// TwinCAT 3 PLC project FMS_201_Estructurado
// ProgramVersion: 3.1.4024.0
// libraries:
//   Tc2_Standard, * (Beckhoff Automation GmbH)
//   Tc2_System, * (Beckhoff Automation GmbH)
//   Tc3_Module, * (Beckhoff Automation GmbH)
// project tree:
//   / PlcTask.TcTTO
//   POUs/Estación/ FB_Coordinador_SFC.TcPOU, FB_Estacion_SFC.TcPOU
//   POUs/ MAIN.TcPOU (not stored)
//   POUs/Tareas/ FB_2_AlimentarBase_SFC.TcPOU (not stored), FB_1_CargarBase_SFC.TcPOU, FB_4_InsertarBasePale_SFCC.TcPOU, FB_5_TransferirBase_SFC.TcPOU, FB_3_VerificarPale_SFC.TcPOU
// (motion and I/O tree: see PLC project fms_201_manual)
// real-time tasks:
//   TASK PlcTask: cycle T#10ms, priority 20, ADS port 350
//   TASK PlcTask1: cycle T#10ms, priority 21, ADS port 351
//   TASK PlcTask2: cycle T#10ms, priority 22, ADS port 352
// variable links:

CONFIGURATION FMS_201_Estructurado
    RESOURCE PLC ON TwinCAT3
        TASK PlcTask(INTERVAL := T#10ms, PRIORITY := 21);
        PROGRAM MAIN WITH PlcTask : MAIN;
    END_RESOURCE
END_CONFIGURATION

// ---- POUs/Estación/FB_Coordinador_SFC.TcPOU
FUNCTION_BLOCK FB_Coordinador_SFC
VAR_INPUT
END_VAR
VAR_OUTPUT
END_VAR
VAR
END_VAR

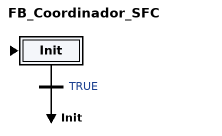
INITIAL_STEP Init:
END_STEP
TRANSITION FROM Init TO Init
    := TRUE;
END_TRANSITION

END_FUNCTION_BLOCK

// ---- POUs/Estación/FB_Estacion_SFC.TcPOU
FUNCTION_BLOCK FB_Estacion_SFC
VAR_INPUT
	// SFC-Flags
	SFCReset: BOOL;
	
	// Parámetros
	TpoEstabilidad: TIME := T#1000MS;
	UdsSolicitadas:UINT := 5;
	
END_VAR
VAR_OUTPUT
	// Parámetros
	CondicionInicial: BOOL;
	UdsPendientes: UINT;
	UdsRealizadas: BOOL;
	
	// Entradas comunes
	PulsadorEmergencia AT %I*: BOOL;
    SelectorManual AT %I*: BOOL;
    PulsadorMarcha AT %I*: BOOL;
    PulsadorParada AT %I*: BOOL := TRUE; // Contacto normalmente cerrado
    EstacionConectada AT %I*: BOOL := TRUE;
    DetectorPresion AT %I*: BOOL := TRUE;
	
	PalePresencia AT %I*: BOOL;
    PaleCodigoBit0 AT %I*: BOOL;
    PaleCodigoBit1 AT %I*: BOOL;
    PaleCodigoBit2 AT %I*: BOOL;
	
	// Entradas específicas
	DescargadorDetras AT %I*: BOOL;
	DescargadorDelante AT %I*: BOOL;
	VerticalArriba AT %I*: BOOL;
	VerticalAbajo AT %I*: BOOL;
	VerificadorArriba AT %I*: BOOL;
	VerificadorAbajo AT %I*: BOOL;
	DesplazadorDetras AT %I*: BOOL;
	AlimentadorDetras AT %I*: BOOL;
	AlimentadorDelante AT %I*: BOOL;
	VacioDescargador AT %I*: BOOL;
	PresenciaBaseAlimentador AT %I*:BOOL;
END_VAR
VAR
	// Bloques funcionales
	CLK: FB_Clock;
	// Salidas comunes
	DesconectaEstacion AT %Q*: BOOL;
    LamparaAlarma AT %Q*: BOOL;
    LamparaMarcha AT %Q*: BOOL;
	LamparaFaltaMaterial AT %Q*: BOOL;
    AvisadorSonoro AT %Q*: BOOL;

    CintaMotorActiva AT %Q*: BOOL;
    CintaMotorInvierte AT %Q*: BOOL;
    CintaRetenedorBaja AT %Q*: BOOL;
    CintaSeparadorSube AT %Q*: BOOL;
	
	// Salidas específicas
	DescargadorAtras AT %Q*: BOOL;
	DescargadorAdelante AT %Q*: BOOL;
	DescargadorBaja AT %Q*: BOOL;
	RechazadorAdelante AT %Q*: BOOL;
	VerificadorBaja AT %Q*: BOOL;
	DesplazadorAdelante AT %Q*: BOOL;
	AlimentadorAdelante AT %Q*: BOOL;
	EyectorSucciona AT %Q*: BOOL;
END_VAR

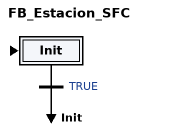
INITIAL_STEP Init:
END_STEP
TRANSITION FROM Init TO Init
    := TRUE;
END_TRANSITION

END_FUNCTION_BLOCK

// ---- POUs/Tareas/FB_1_CargarBase_SFC.TcPOU
FUNCTION_BLOCK FB_1_CargarBase_SFC
VAR_INPUT
	
	// Indicadores de sincronización
	Ack: BOOL := TRUE;
	Execute: BOOL;
	
	// Entradas
	PalePresencia AT %I*: BOOL;
	
END_VAR
VAR_OUTPUT
	
	// Indicadores de sincronización
	Ready: BOOL;	
	Done: BOOL;
	
	// Salidas
	CintaMotorActiva AT %Q*: BOOL;
	
END_VAR
VAR
END_VAR

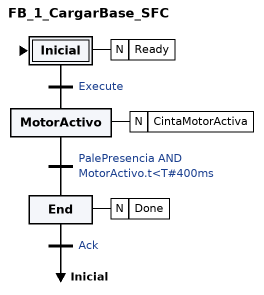
INITIAL_STEP Inicial:
    Ready(N);
END_STEP
TRANSITION FROM Inicial TO MotorActivo
    := Execute;
END_TRANSITION
STEP MotorActivo:
    CintaMotorActiva(N);
END_STEP
TRANSITION FROM MotorActivo TO End
    := PalePresencia AND MotorActivo.t<T#400ms;
END_TRANSITION
STEP End:
    Done(N);
END_STEP
TRANSITION FROM End TO Inicial
    := Ack;
END_TRANSITION

END_FUNCTION_BLOCK

// ---- POUs/Tareas/FB_4_InsertarBasePale_SFCC.TcPOU
FUNCTION_BLOCK FB_4_InsertarBasePale_SFCC
VAR_INPUT

// Indicadores de sincronización
	Ack: BOOL := TRUE;
	Execute: BOOL;
	
	// Parámetros
	TpoTraspase: TIME := T#500MS;
	
	// Entradas
	VerticalArriba AT %I*: BOOL;
	VerticalAbajo AT %I*: BOOL;
	VacioDescargador AT %I*: BOOL;	
	DescargadorDetras AT %I*: BOOL;
	DescargadorDelante AT %I*: BOOL;
	
END_VAR
VAR_OUTPUT
	
// Indicadores de sincronización
	Ready: BOOL;	
	Done: BOOL;
	
	// Salidas
	DescargadorAtras AT %Q*: BOOL;
	DescargadorAdelante AT %Q*: BOOL;
	DescargadorBaja AT %Q*: BOOL;
	EyectorSucciona AT %Q*: BOOL;
	
END_VAR
VAR
END_VAR

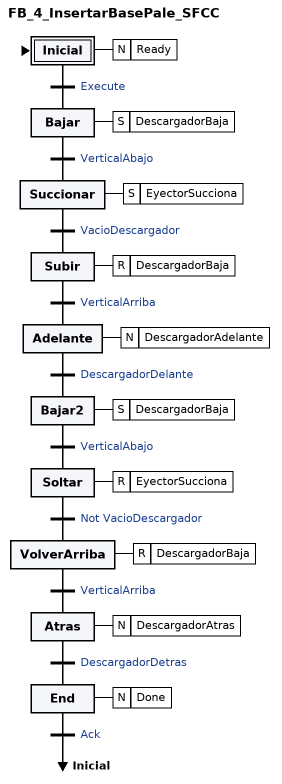
INITIAL_STEP Inicial:
    Ready(N);
END_STEP
TRANSITION FROM Inicial TO Bajar
    := Execute;
END_TRANSITION
STEP Bajar:
    DescargadorBaja(S);
END_STEP
TRANSITION FROM Bajar TO Succionar
    := VerticalAbajo;
END_TRANSITION
STEP Succionar:
    EyectorSucciona(S);
END_STEP
TRANSITION FROM Succionar TO Subir
    := VacioDescargador;
END_TRANSITION
STEP Subir:
    DescargadorBaja(R);
END_STEP
TRANSITION FROM Subir TO Adelante
    := VerticalArriba;
END_TRANSITION
STEP Adelante:
    DescargadorAdelante(N);
END_STEP
TRANSITION FROM Adelante TO Bajar2
    := DescargadorDelante;
END_TRANSITION
STEP Bajar2:
    DescargadorBaja(S);
END_STEP
TRANSITION FROM Bajar2 TO Soltar
    := VerticalAbajo;
END_TRANSITION
STEP Soltar:
    EyectorSucciona(R);
END_STEP
TRANSITION FROM Soltar TO VolverArriba
    := Not VacioDescargador;
END_TRANSITION
STEP VolverArriba:
    DescargadorBaja(R);
END_STEP
TRANSITION FROM VolverArriba TO Atras
    := VerticalArriba;
END_TRANSITION
STEP Atras:
    DescargadorAtras(N);
END_STEP
TRANSITION FROM Atras TO End
    := DescargadorDetras;
END_TRANSITION
STEP End:
    Done(N);
END_STEP
TRANSITION FROM End TO Inicial
    := Ack;
END_TRANSITION

END_FUNCTION_BLOCK

// ---- POUs/Tareas/FB_5_TransferirBase_SFC.TcPOU
FUNCTION_BLOCK FB_5_TransferirBase_SFC
VAR_INPUT
	
	// Indicadores de sincronización
	Ack: BOOL := TRUE;
	Execute: BOOL;
	
	// Parámetros
	TpoBasesALE: TIME := T#500MS;
	
	// Entradas
	PalePresencia: BOOL;
	
END_VAR
VAR_OUTPUT
	
	// Indicadores de sincronización
	Ready: BOOL;	
	Done: BOOL;
	
	// Salidas
	CintaMotorActiva: BOOL;
	CintaRetenedorBaja: BOOL;
	CintaSeparadorSube: BOOL;
	
END_VAR
VAR
END_VAR

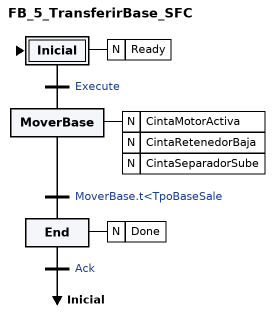
INITIAL_STEP Inicial:
    Ready(N);
END_STEP
TRANSITION FROM Inicial TO MoverBase
    := Execute;
END_TRANSITION
STEP MoverBase:
    CintaMotorActiva(N);
    CintaRetenedorBaja(N);
    CintaSeparadorSube(N);
END_STEP
TRANSITION FROM MoverBase TO End
    := MoverBase.t<TpoBaseSale;
END_TRANSITION
STEP End:
    Done(N);
END_STEP
TRANSITION FROM End TO Inicial
    := Ack;
END_TRANSITION

END_FUNCTION_BLOCK

// ---- POUs/Tareas/FB_3_VerificarPale_SFC.TcPOU
FUNCTION_BLOCK FB_3_VerificarPale_SFC
VAR_INPUT
	
	// Indicadores de sincronización
	Ack: BOOL := TRUE;
	Execute: BOOL;
	
	// Entradas
	VerificadorAbajo: BOOL;
	VerificadorArriba: BOOL;
	DesplazadorDetras: BOOL;
	
	
END_VAR
VAR_OUTPUT
	
	// Indicadores de sincronización
	Ready: BOOL;	
	Done: BOOL;
	
	// Salidas
	VerificadorBaja: BOOL;
	DesplazadorAdelante: BOOL;
	RechazadorAdelante: BOOL;
	
END_VAR

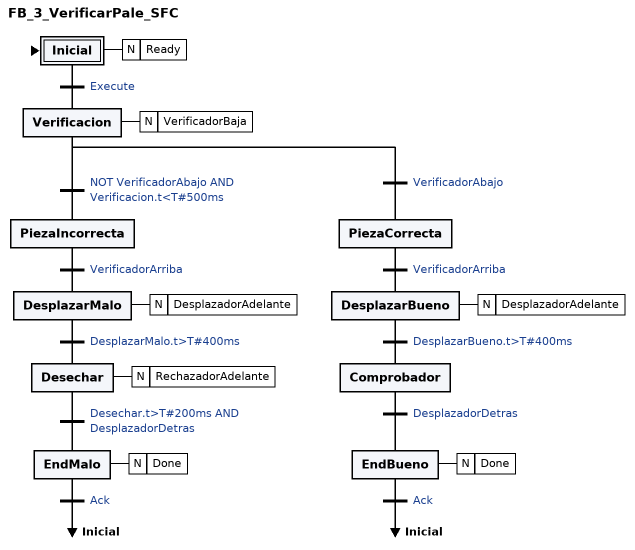
INITIAL_STEP Inicial:
    Ready(N);
END_STEP
TRANSITION FROM Inicial TO Verificacion
    := Execute;
END_TRANSITION
STEP Verificacion:
    VerificadorBaja(N);
END_STEP
TRANSITION FROM Verificacion TO PiezaIncorrecta
    := NOT VerificadorAbajo AND Verificacion.t<T#500ms;
END_TRANSITION
STEP PiezaIncorrecta:
END_STEP
TRANSITION FROM PiezaIncorrecta TO DesplazarMalo
    := VerificadorArriba;
END_TRANSITION
STEP DesplazarMalo:
    DesplazadorAdelante(N);
END_STEP
TRANSITION FROM DesplazarMalo TO Desechar
    := DesplazarMalo.t>T#400ms;
END_TRANSITION
STEP Desechar:
    RechazadorAdelante(N);
END_STEP
TRANSITION FROM Desechar TO EndMalo
    := Desechar.t>T#200ms AND DesplazadorDetras;
END_TRANSITION
STEP EndMalo:
    Done(N);
END_STEP
TRANSITION FROM EndMalo TO Inicial
    := Ack;
END_TRANSITION
TRANSITION FROM Verificacion TO PiezaCorrecta
    := VerificadorAbajo;
END_TRANSITION
STEP PiezaCorrecta:
END_STEP
TRANSITION FROM PiezaCorrecta TO DesplazarBueno
    := VerificadorArriba;
END_TRANSITION
STEP DesplazarBueno:
    DesplazadorAdelante(N);
END_STEP
TRANSITION FROM DesplazarBueno TO Comprobador
    := DesplazarBueno.t>T#400ms;
END_TRANSITION
STEP Comprobador:
END_STEP
TRANSITION FROM Comprobador TO EndBueno
    := DesplazadorDetras;
END_TRANSITION
STEP EndBueno:
    Done(N);
END_STEP
TRANSITION FROM EndBueno TO Inicial
    := Ack;
END_TRANSITION

END_FUNCTION_BLOCK
